{attribute 'linkalways'} 
{attribute 'no_explicit_call' := 'This FB is a CLASS and must be accessed using methods or properties'}
{attribute 'enable_dynamic_creation'}
FUNCTION_BLOCK RegisterInstanceToTaskCallback IMPLEMENTS I_Callback
VAR
	task : I_Task;
END_VAR

METHOD FB_init : BOOL
VAR_INPUT
	bInitRetains : BOOL; // if TRUE, the retain variables are initialized (warm start / cold start)
	bInCopyCode : BOOL;  // if TRUE, the instance afterwards gets moved into the copy code (online change)
	Task : I_Task;
END_VAR
this^.task := Task;
END_METHOD

METHOD PUBLIC Update
VAR_INPUT
	event : I_Event;
END_VAR
VAR
	instanceAdded : I_InstanceAddedEvent;
END_VAR
IF NOT __QUERYINTERFACE(event, instanceAdded) THEN
	RETURN;
END_IF

IF task.SharesNamespaceWith(instanceAdded.Instance) THEN
	task.RegisterInstance(instanceAdded.Instance);
	RETURN;
END_IF

IF task.IsExecutingThis() THEN
	task.RegisterInstance(instanceAdded.Instance);
	RETURN;
END_IF
END_METHOD

END_FUNCTION_BLOCK

(* stored: Version 1.1.0.1, ProductVersion 3.1.4024.12
   POU RegisterInstanceToTaskCallback: Id {59905fa2-13da-00cb-0d49-56c42ae3a073}, SpecialFunc None
   Folder Constructor: Id {9c2f0530-da68-02f0-231e-8885d07d78f3}
   Method FB_init: Id {b952bc26-687a-0b7a-10ff-62034c799119}
   Method Update: Id {5b4f5c4c-aa4e-00e8-3a56-bf226c8af173} *)
